// Builds a Sparkplug B DDEATH payload.
//
// DDEATH announces that a logical device is going offline. It carries only a
// timestamp and seq — no metrics. The session manager publishes it before
// disconnecting a device or on detecting a device fault.
FUNCTION_BLOCK FB_DDeathBuilder
VAR
	_aBuf		: ARRAY[0..31] OF BYTE;
	_fbPayload	: FB_SparkplugPayload;
END_VAR

// FB body intentionally empty — all logic is in Build().

METHOD Build : BOOL
VAR_INPUT
	nTimestamp	: ULINT;
	nSeq		: ULINT;
END_VAR
_fbPayload.Init(ADR(_aBuf), SIZEOF(_aBuf));
_fbPayload.WriteHeader(nTimestamp, nSeq);
Build := NOT _fbPayload.HasError;
END_METHOD

PROPERTY Payload : REFERENCE TO FB_SparkplugPayload
GET
Payload REF= _fbPayload;
END_GET
END_PROPERTY

END_FUNCTION_BLOCK

(* stored: Version 1.1.0.1
   POU FB_DDeathBuilder: Id {66666666-7777-8888-9999-aaaaaaaaaaaa}, SpecialFunc None
   Method Build: Id {77777777-8888-9999-aaaa-bbbbbbbbbbbb}
   Property Payload: Id {88888888-9999-aaaa-bbbb-cccccccccccc}
   Get Get: Id {99999999-aaaa-bbbb-cccc-dddddddddddd} *)
